FUNCTION_BLOCK FB_WearPart
VAR_INPUT
localClock : DATE_AND_TIME; //
END_VAR
VAR_IN_OUT
machine : UDT_Machine_RD; //
stations : UDT_Station_RD; //
vari : UDT_WearPartVar_RD; //
data : UDT_WearPartData_RD; //
END_VAR
VAR
nIndex : UINT;
tipTimes : DINT;//提示次数             
END_VAR

Execute();
Alarm();
Clear();

ACTION Alarm:
tipTimes:=LREAL_TO_DINT(DINT_TO_LREAL(data.maxUsage)*REAL_TO_LREAL(data.tipRate)/100);


vari.alarming:=data.actUsage>=data.maxUsage;
vari.tip:=data.actUsage>=tipTimes AND NOT vari.alarming;
END_ACTION

ACTION Clear:
vari.clearHmi :=
vari.clearAuto := FALSE;
IF data.actUsage>0 THEN
  vari.clearAllow:=vari.clearPermit;
  IF vari.clearAllow AND machine.manualMode THEN
      vari.clearForbidIcon := NOT vari.clearAllow;//清零禁止图标
      IF vari.clearAllow AND (vari.clearHmi OR  vari.clearAuto) THEN
        FOR nIndex:=9 TO 1 BY -1 DO
  		  data.recordsTime[nIndex]:=data.recordsTime[nIndex-1];
  		  data.recordsUsage[nIndex]:=data.recordsUsage[nIndex-1];
  	    END_FOR
  	    data.recordsTime[0]:=DT_TO_SYSTEMTIME(localClock);
  	    data.recordsUsage[0]:=data.actUsage;
  	    data.actUsage:=0;
      END_IF;
  ELSE
    vari.clearForbidIcon := TRUE;
  END_IF;
END_IF
END_ACTION

ACTION Execute:
vari.countExecute:=FALSE;
IF vari.countExecute THEN
	data.actUsage:=data.actUsage+vari.increments;
END_IF
END_ACTION

END_FUNCTION_BLOCK

(* stored: Version 1.1.0.1, ProductVersion 3.1.4024.12
   POU FB_WearPart: Id {6a533d51-1840-4ee3-a6bd-679d26e5b4f6}, SpecialFunc None
   Action Alarm: Id {3c55bf18-fcca-4ae5-95d2-b5d7ff80b304}
   Action Clear: Id {c3f06054-4474-4c02-ab07-8bb709dd91e4}
   Action Execute: Id {22f269b0-68b1-44ab-a81a-5b39a0846e1b} *)
